SYSTEM furnace_naphtha_cracker
  (* Version 1.0, 2021-03-12, Lenovo *)
  APPLICATION furnace_naphtha_crackerApp
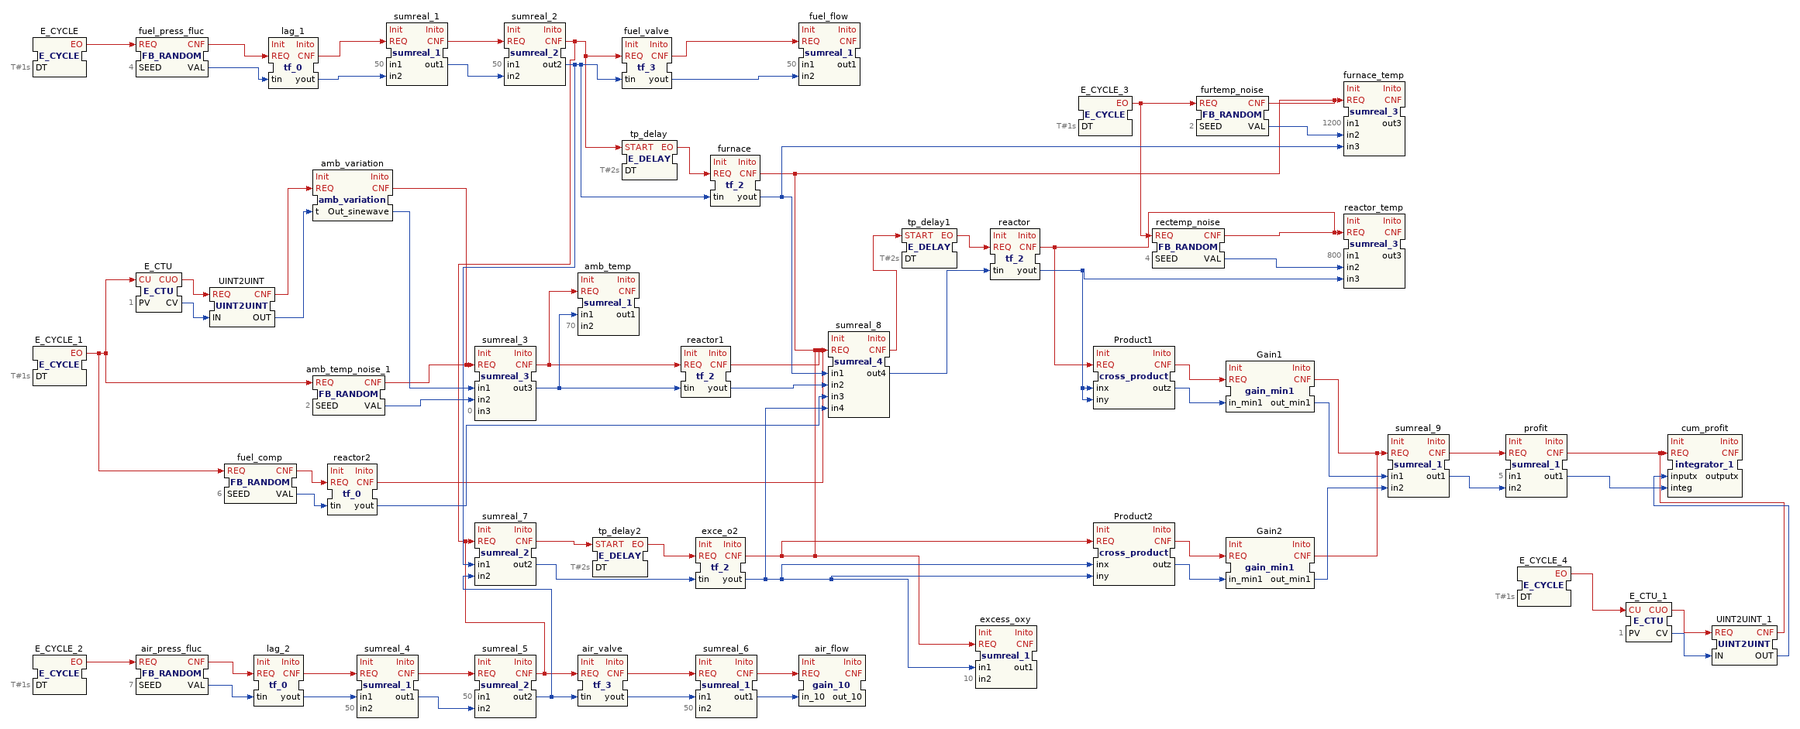
    FBS
      E_CYCLE : E_CYCLE(DT := T#1s);
      sumreal_1 : sumreal_1(in1 := 50);
      sumreal_2 : sumreal_2(in1 := 50);
      fuel_valve : tf_3;
      fuel_flow : sumreal_1(in1 := 50);
      E_CYCLE_1 : E_CYCLE(DT := T#1s);
      E_CTU : E_CTU(PV := 1);
      UINT2UINT : UINT2UINT;
      amb_variation : amb_variation;
      amb_temp_noise_1 : FB_RANDOM(SEED := 2);
      E_CYCLE_2 : E_CYCLE(DT := T#1s);
      air_press_fluc : FB_RANDOM(SEED := 7);
      lag_2 : tf_0;
      sumreal_4 : sumreal_1(in2 := 50);
      sumreal_5 : sumreal_2(in1 := 50);
      air_valve : tf_3;
      sumreal_6 : sumreal_1(in2 := 50);
      air_flow : gain_10;
      reactor1 : tf_2;
      fuel_comp : FB_RANDOM(SEED := 6);
      reactor2 : tf_0;
      sumreal_7 : sumreal_2;
      exce_o2 : tf_2;
      tp_delay : E_DELAY(DT := T#2s);
      furnace : tf_2;
      tp_delay2 : E_DELAY(DT := T#2s);
      sumreal_8 : sumreal_4;
      tp_delay1 : E_DELAY(DT := T#2s);
      reactor : tf_2;
      Product2 : cross_product;
      Gain2 : gain_min1;
      Product1 : cross_product;
      Gain1 : gain_min1;
      sumreal_9 : sumreal_1;
      E_CYCLE_3 : E_CYCLE(DT := T#1s);
      furtemp_noise : FB_RANDOM(SEED := 2);
      rectemp_noise : FB_RANDOM(SEED := 4);
      furnace_temp : sumreal_3(in1 := 1200);
      reactor_temp : sumreal_3(in1 := 800);
      profit : sumreal_1(in1 := 5);
      excess_oxy : sumreal_1(in2 := 10);
      E_CYCLE_4 : E_CYCLE(DT := T#1s);
      E_CTU_1 : E_CTU(PV := 1);
      UINT2UINT_1 : UINT2UINT;
      fuel_press_fluc : FB_RANDOM(SEED := 4);
      lag_1 : tf_0;
      sumreal_3 : sumreal_3(in3 := 0);
      amb_temp : sumreal_1(in2 := 70);
      cum_profit : integrator_1;
    END_FBS
    EVENT_CONNECTIONS
      sumreal_2.CNF TO fuel_valve.REQ;
      sumreal_1.CNF TO sumreal_2.REQ;
      fuel_valve.CNF TO fuel_flow.REQ;
      E_CYCLE_1.EO TO E_CTU.CU;
      E_CTU.CUO TO UINT2UINT.REQ;
      UINT2UINT.CNF TO amb_variation.REQ;
      E_CYCLE_1.EO TO amb_temp_noise_1.REQ;
      E_CYCLE_2.EO TO air_press_fluc.REQ;
      air_press_fluc.CNF TO lag_2.REQ;
      lag_2.CNF TO sumreal_4.REQ;
      sumreal_4.CNF TO sumreal_5.REQ;
      sumreal_5.CNF TO air_valve.REQ;
      air_valve.CNF TO sumreal_6.REQ;
      sumreal_6.CNF TO air_flow.REQ;
      E_CYCLE_1.EO TO fuel_comp.REQ;
      fuel_comp.CNF TO reactor2.REQ;
      sumreal_5.CNF TO sumreal_7.REQ;
      sumreal_2.CNF TO sumreal_7.REQ;
      sumreal_2.CNF TO tp_delay.START;
      tp_delay.EO TO furnace.REQ;
      sumreal_7.CNF TO tp_delay2.START;
      tp_delay2.EO TO exce_o2.REQ;
      furnace.CNF TO sumreal_8.REQ;
      reactor1.CNF TO sumreal_8.REQ;
      exce_o2.CNF TO sumreal_8.REQ;
      reactor2.CNF TO sumreal_8.REQ;
      sumreal_8.CNF TO tp_delay1.START;
      tp_delay1.EO TO reactor.REQ;
      exce_o2.CNF TO Product2.REQ;
      Product2.CNF TO Gain2.REQ;
      Product1.CNF TO Gain1.REQ;
      Gain1.CNF TO sumreal_9.REQ;
      Gain2.CNF TO sumreal_9.REQ;
      E_CYCLE_3.EO TO furtemp_noise.REQ;
      furnace.CNF TO furnace_temp.REQ;
      furtemp_noise.CNF TO furnace_temp.REQ;
      E_CYCLE_3.EO TO rectemp_noise.REQ;
      rectemp_noise.CNF TO reactor_temp.REQ;
      reactor.CNF TO Product1.REQ;
      reactor.CNF TO reactor_temp.REQ;
      sumreal_9.CNF TO profit.REQ;
      exce_o2.CNF TO excess_oxy.REQ;
      E_CTU_1.CUO TO UINT2UINT_1.REQ;
      E_CYCLE_4.EO TO E_CTU_1.CU;
      lag_1.CNF TO sumreal_1.REQ;
      E_CYCLE.EO TO fuel_press_fluc.REQ;
      fuel_press_fluc.CNF TO lag_1.REQ;
      sumreal_3.CNF TO reactor1.REQ;
      amb_temp_noise_1.CNF TO sumreal_3.REQ;
      amb_variation.CNF TO sumreal_3.REQ;
      sumreal_3.CNF TO amb_temp.REQ;
      profit.CNF TO cum_profit.REQ;
      UINT2UINT_1.CNF TO cum_profit.REQ;
    END_CONNECTIONS
    DATA_CONNECTIONS
      sumreal_1.out1 TO sumreal_2.in2;
      sumreal_2.out2 TO fuel_valve.tin;
      fuel_valve.yout TO fuel_flow.in2;
      E_CTU.CV TO UINT2UINT.IN;
      UINT2UINT.OUT TO amb_variation.t;
      air_press_fluc.VAL TO lag_2.tin;
      lag_2.yout TO sumreal_4.in1;
      sumreal_4.out1 TO sumreal_5.in2;
      sumreal_5.out2 TO air_valve.tin;
      air_valve.yout TO sumreal_6.in1;
      sumreal_6.out1 TO air_flow.in_10;
      fuel_comp.VAL TO reactor2.tin;
      sumreal_5.out2 TO sumreal_7.in2;
      sumreal_2.out2 TO sumreal_7.in1;
      sumreal_7.out2 TO exce_o2.tin;
      sumreal_2.out2 TO furnace.tin;
      furnace.yout TO sumreal_8.in1;
      reactor1.yout TO sumreal_8.in2;
      exce_o2.yout TO sumreal_8.in4;
      reactor2.yout TO sumreal_8.in3;
      sumreal_8.out4 TO reactor.tin;
      exce_o2.yout TO Product2.inx;
      exce_o2.yout TO Product2.iny;
      Product2.outz TO Gain2.in_min1;
      Product1.outz TO Gain1.in_min1;
      reactor.yout TO Product1.inx;
      reactor.yout TO Product1.iny;
      Gain2.out_min1 TO sumreal_9.in2;
      Gain1.out_min1 TO sumreal_9.in1;
      furtemp_noise.VAL TO furnace_temp.in2;
      furnace.yout TO furnace_temp.in3;
      rectemp_noise.VAL TO reactor_temp.in2;
      reactor.yout TO reactor_temp.in3;
      sumreal_9.out1 TO profit.in2;
      exce_o2.yout TO excess_oxy.in1;
      E_CTU_1.CV TO UINT2UINT_1.IN;
      lag_1.yout TO sumreal_1.in2;
      fuel_press_fluc.VAL TO lag_1.tin;
      sumreal_3.out3 TO reactor1.tin;
      amb_temp_noise_1.VAL TO sumreal_3.in2;
      amb_variation.Out_sinewave TO sumreal_3.in1;
      sumreal_3.out3 TO amb_temp.in1;
      UINT2UINT_1.OUT TO cum_profit.inputx;
      profit.out1 TO cum_profit.integ;
    END_CONNECTIONS
  END_APPLICATION
  DEVICE FORTE_PC : FORTE_PC(MGR_ID := "localhost:61499")
    {SET_ATTRIBUTE(Profile, HOLOBLOC)} (* device profile *)
    RESOURCE EMB_RES : EMB_RES
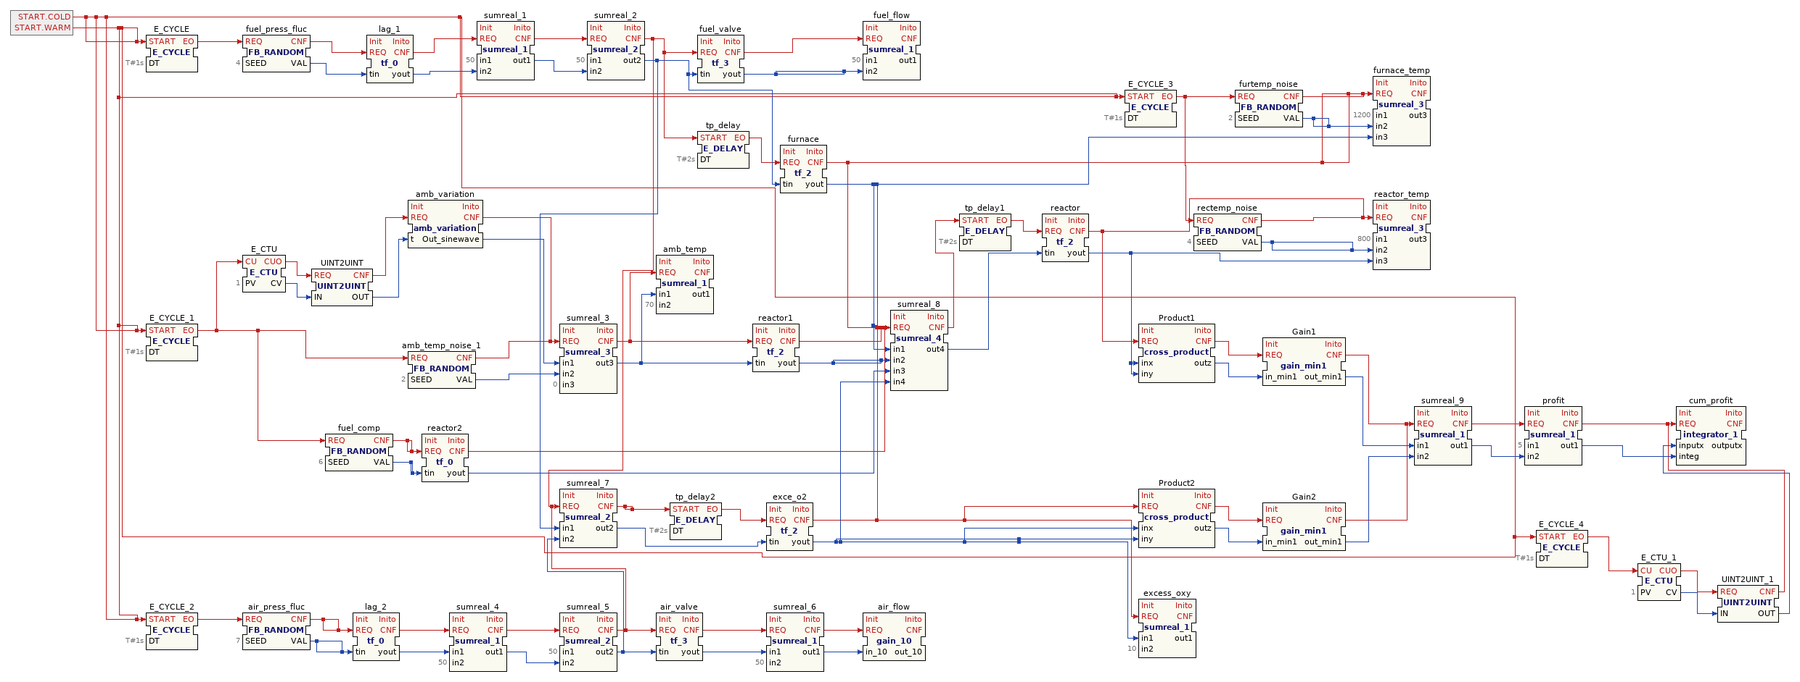
      FBS
        fuel_valve : tf_3;
        fuel_flow : sumreal_1(in1 := 50);
        E_CYCLE_1 : E_CYCLE(DT := T#1s);
        E_CTU : E_CTU(PV := 1);
        UINT2UINT : UINT2UINT;
        amb_variation : amb_variation;
        amb_temp_noise_1 : FB_RANDOM(SEED := 2);
        E_CYCLE_2 : E_CYCLE(DT := T#1s);
        air_press_fluc : FB_RANDOM(SEED := 7);
        lag_2 : tf_0;
        sumreal_4 : sumreal_1(in2 := 50);
        sumreal_5 : sumreal_2(in1 := 50);
        air_valve : tf_3;
        sumreal_6 : sumreal_1(in2 := 50);
        air_flow : gain_10;
        reactor1 : tf_2;
        fuel_comp : FB_RANDOM(SEED := 6);
        reactor2 : tf_0;
        sumreal_7 : sumreal_2;
        exce_o2 : tf_2;
        tp_delay : E_DELAY(DT := T#2s);
        furnace : tf_2;
        tp_delay2 : E_DELAY(DT := T#2s);
        sumreal_8 : sumreal_4;
        tp_delay1 : E_DELAY(DT := T#2s);
        reactor : tf_2;
        Product2 : cross_product;
        Gain2 : gain_min1;
        Product1 : cross_product;
        Gain1 : gain_min1;
        sumreal_9 : sumreal_1;
        E_CYCLE_3 : E_CYCLE(DT := T#1s);
        furtemp_noise : FB_RANDOM(SEED := 2);
        rectemp_noise : FB_RANDOM(SEED := 4);
        furnace_temp : sumreal_3(in1 := 1200);
        reactor_temp : sumreal_3(in1 := 800);
        profit : sumreal_1(in1 := 5);
        excess_oxy : sumreal_1(in2 := 10);
        E_CYCLE_4 : E_CYCLE(DT := T#1s);
        E_CTU_1 : E_CTU(PV := 1);
        UINT2UINT_1 : UINT2UINT;
        E_CYCLE : E_CYCLE(DT := T#1s);
        sumreal_1 : sumreal_1(in1 := 50);
        sumreal_2 : sumreal_2(in1 := 50);
        fuel_valve : tf_3;
        fuel_flow : sumreal_1(in1 := 50);
        E_CYCLE_1 : E_CYCLE(DT := T#1s);
        E_CTU : E_CTU(PV := 1);
        UINT2UINT : UINT2UINT;
        amb_variation : amb_variation;
        amb_temp_noise_1 : FB_RANDOM(SEED := 2);
        E_CYCLE_2 : E_CYCLE(DT := T#1s);
        air_press_fluc : FB_RANDOM(SEED := 7);
        lag_2 : tf_0;
        sumreal_4 : sumreal_1(in2 := 50);
        sumreal_5 : sumreal_2(in1 := 50);
        air_valve : tf_3;
        sumreal_6 : sumreal_1(in2 := 50);
        air_flow : gain_10;
        reactor1 : tf_2;
        fuel_comp : FB_RANDOM(SEED := 6);
        reactor2 : tf_0;
        sumreal_7 : sumreal_2;
        exce_o2 : tf_2;
        tp_delay : E_DELAY(DT := T#2s);
        furnace : tf_2;
        tp_delay2 : E_DELAY(DT := T#2s);
        sumreal_8 : sumreal_4;
        tp_delay1 : E_DELAY(DT := T#2s);
        reactor : tf_2;
        Product2 : cross_product;
        Gain2 : gain_min1;
        Product1 : cross_product;
        Gain1 : gain_min1;
        sumreal_9 : sumreal_1;
        E_CYCLE_3 : E_CYCLE(DT := T#1s);
        furtemp_noise : FB_RANDOM(SEED := 2);
        rectemp_noise : FB_RANDOM(SEED := 4);
        furnace_temp : sumreal_3(in1 := 1200);
        reactor_temp : sumreal_3(in1 := 800);
        profit : sumreal_1(in1 := 5);
        excess_oxy : sumreal_1(in2 := 10);
        E_CYCLE_4 : E_CYCLE(DT := T#1s);
        E_CTU_1 : E_CTU(PV := 1);
        UINT2UINT_1 : UINT2UINT;
        fuel_press_fluc : FB_RANDOM(SEED := 4);
        lag_1 : tf_0;
        sumreal_3 : sumreal_3(in3 := 0);
        amb_temp : sumreal_1(in2 := 70);
        cum_profit : integrator_1;
        sumreal_2 : sumreal_2(in1 := 50);
        sumreal_1 : sumreal_1(in1 := 50);
        E_CYCLE : E_CYCLE(DT := T#1s);
      END_FBS
      EVENT_CONNECTIONS
        fuel_valve.CNF TO fuel_flow.REQ;
        E_CYCLE_1.EO TO E_CTU.CU;
        E_CTU.CUO TO UINT2UINT.REQ;
        UINT2UINT.CNF TO amb_variation.REQ;
        E_CYCLE_1.EO TO amb_temp_noise_1.REQ;
        E_CYCLE_2.EO TO air_press_fluc.REQ;
        air_press_fluc.CNF TO lag_2.REQ;
        lag_2.CNF TO sumreal_4.REQ;
        sumreal_4.CNF TO sumreal_5.REQ;
        sumreal_5.CNF TO air_valve.REQ;
        air_valve.CNF TO sumreal_6.REQ;
        sumreal_6.CNF TO air_flow.REQ;
        E_CYCLE_1.EO TO fuel_comp.REQ;
        fuel_comp.CNF TO reactor2.REQ;
        sumreal_5.CNF TO sumreal_7.REQ;
        tp_delay.EO TO furnace.REQ;
        sumreal_7.CNF TO tp_delay2.START;
        tp_delay2.EO TO exce_o2.REQ;
        furnace.CNF TO sumreal_8.REQ;
        reactor1.CNF TO sumreal_8.REQ;
        exce_o2.CNF TO sumreal_8.REQ;
        reactor2.CNF TO sumreal_8.REQ;
        sumreal_8.CNF TO tp_delay1.START;
        tp_delay1.EO TO reactor.REQ;
        exce_o2.CNF TO Product2.REQ;
        Product2.CNF TO Gain2.REQ;
        reactor.CNF TO Product1.REQ;
        Product1.CNF TO Gain1.REQ;
        Gain1.CNF TO sumreal_9.REQ;
        Gain2.CNF TO sumreal_9.REQ;
        E_CYCLE_3.EO TO furtemp_noise.REQ;
        E_CYCLE_3.EO TO rectemp_noise.REQ;
        furnace.CNF TO furnace_temp.REQ;
        furtemp_noise.CNF TO furnace_temp.REQ;
        rectemp_noise.CNF TO reactor_temp.REQ;
        reactor.CNF TO reactor_temp.REQ;
        sumreal_9.CNF TO profit.REQ;
        exce_o2.CNF TO excess_oxy.REQ;
        E_CYCLE_4.EO TO E_CTU_1.CU;
        E_CTU_1.CUO TO UINT2UINT_1.REQ;
        sumreal_1.CNF TO sumreal_2.REQ;
        sumreal_2.CNF TO fuel_valve.REQ;
        fuel_valve.CNF TO fuel_flow.REQ;
        E_CYCLE_1.EO TO E_CTU.CU;
        E_CTU.CUO TO UINT2UINT.REQ;
        UINT2UINT.CNF TO amb_variation.REQ;
        E_CYCLE_1.EO TO amb_temp_noise_1.REQ;
        E_CYCLE_2.EO TO air_press_fluc.REQ;
        air_press_fluc.CNF TO lag_2.REQ;
        lag_2.CNF TO sumreal_4.REQ;
        sumreal_4.CNF TO sumreal_5.REQ;
        sumreal_5.CNF TO air_valve.REQ;
        air_valve.CNF TO sumreal_6.REQ;
        sumreal_6.CNF TO air_flow.REQ;
        E_CYCLE_1.EO TO fuel_comp.REQ;
        fuel_comp.CNF TO reactor2.REQ;
        sumreal_5.CNF TO sumreal_7.REQ;
        sumreal_2.CNF TO sumreal_7.REQ;
        sumreal_2.CNF TO tp_delay.START;
        tp_delay.EO TO furnace.REQ;
        sumreal_7.CNF TO tp_delay2.START;
        tp_delay2.EO TO exce_o2.REQ;
        furnace.CNF TO sumreal_8.REQ;
        reactor1.CNF TO sumreal_8.REQ;
        exce_o2.CNF TO sumreal_8.REQ;
        reactor2.CNF TO sumreal_8.REQ;
        sumreal_8.CNF TO tp_delay1.START;
        tp_delay1.EO TO reactor.REQ;
        exce_o2.CNF TO Product2.REQ;
        Product2.CNF TO Gain2.REQ;
        reactor.CNF TO Product1.REQ;
        Product1.CNF TO Gain1.REQ;
        Gain1.CNF TO sumreal_9.REQ;
        Gain2.CNF TO sumreal_9.REQ;
        E_CYCLE_3.EO TO furtemp_noise.REQ;
        E_CYCLE_3.EO TO rectemp_noise.REQ;
        furnace.CNF TO furnace_temp.REQ;
        furtemp_noise.CNF TO furnace_temp.REQ;
        rectemp_noise.CNF TO reactor_temp.REQ;
        reactor.CNF TO reactor_temp.REQ;
        sumreal_9.CNF TO profit.REQ;
        exce_o2.CNF TO excess_oxy.REQ;
        E_CYCLE_4.EO TO E_CTU_1.CU;
        E_CTU_1.CUO TO UINT2UINT_1.REQ;
        E_CYCLE.EO TO fuel_press_fluc.REQ;
        fuel_press_fluc.CNF TO lag_1.REQ;
        lag_1.CNF TO sumreal_1.REQ;
        amb_temp_noise_1.CNF TO sumreal_3.REQ;
        amb_variation.CNF TO sumreal_3.REQ;
        sumreal_3.CNF TO reactor1.REQ;
        sumreal_3.CNF TO amb_temp.REQ;
        profit.CNF TO cum_profit.REQ;
        UINT2UINT_1.CNF TO cum_profit.REQ;
        START.COLD TO E_CYCLE.START;
        START.WARM TO E_CYCLE.START;
        START.COLD TO E_CYCLE_1.START;
        START.WARM TO E_CYCLE_1.START;
        START.COLD TO E_CYCLE_2.START;
        START.WARM TO E_CYCLE_2.START;
        START.COLD TO E_CYCLE_4.START;
        START.WARM TO E_CYCLE_4.START;
        START.COLD TO E_CYCLE_3.START;
        START.WARM TO E_CYCLE_3.START;
        sumreal_2.CNF TO tp_delay.START;
        sumreal_2.CNF TO sumreal_7.REQ;
        sumreal_2.CNF TO fuel_valve.REQ;
        sumreal_1.CNF TO sumreal_2.REQ;
      END_CONNECTIONS
      DATA_CONNECTIONS
        fuel_valve.yout TO fuel_flow.in2;
        E_CTU.CV TO UINT2UINT.IN;
        UINT2UINT.OUT TO amb_variation.t;
        air_press_fluc.VAL TO lag_2.tin;
        lag_2.yout TO sumreal_4.in1;
        sumreal_4.out1 TO sumreal_5.in2;
        sumreal_5.out2 TO air_valve.tin;
        air_valve.yout TO sumreal_6.in1;
        sumreal_6.out1 TO air_flow.in_10;
        fuel_comp.VAL TO reactor2.tin;
        sumreal_5.out2 TO sumreal_7.in2;
        sumreal_7.out2 TO exce_o2.tin;
        furnace.yout TO sumreal_8.in1;
        reactor1.yout TO sumreal_8.in2;
        reactor2.yout TO sumreal_8.in3;
        exce_o2.yout TO sumreal_8.in4;
        sumreal_8.out4 TO reactor.tin;
        exce_o2.yout TO Product2.inx;
        exce_o2.yout TO Product2.iny;
        Product2.outz TO Gain2.in_min1;
        reactor.yout TO Product1.inx;
        reactor.yout TO Product1.iny;
        Product1.outz TO Gain1.in_min1;
        Gain1.out_min1 TO sumreal_9.in1;
        Gain2.out_min1 TO sumreal_9.in2;
        furtemp_noise.VAL TO furnace_temp.in2;
        furnace.yout TO furnace_temp.in3;
        rectemp_noise.VAL TO reactor_temp.in2;
        reactor.yout TO reactor_temp.in3;
        sumreal_9.out1 TO profit.in2;
        exce_o2.yout TO excess_oxy.in1;
        E_CTU_1.CV TO UINT2UINT_1.IN;
        sumreal_1.out1 TO sumreal_2.in2;
        sumreal_2.out2 TO fuel_valve.tin;
        fuel_valve.yout TO fuel_flow.in2;
        E_CTU.CV TO UINT2UINT.IN;
        UINT2UINT.OUT TO amb_variation.t;
        air_press_fluc.VAL TO lag_2.tin;
        lag_2.yout TO sumreal_4.in1;
        sumreal_4.out1 TO sumreal_5.in2;
        sumreal_5.out2 TO air_valve.tin;
        air_valve.yout TO sumreal_6.in1;
        sumreal_6.out1 TO air_flow.in_10;
        fuel_comp.VAL TO reactor2.tin;
        sumreal_2.out2 TO sumreal_7.in1;
        sumreal_5.out2 TO sumreal_7.in2;
        sumreal_7.out2 TO exce_o2.tin;
        sumreal_2.out2 TO furnace.tin;
        furnace.yout TO sumreal_8.in1;
        reactor1.yout TO sumreal_8.in2;
        reactor2.yout TO sumreal_8.in3;
        exce_o2.yout TO sumreal_8.in4;
        sumreal_8.out4 TO reactor.tin;
        exce_o2.yout TO Product2.inx;
        exce_o2.yout TO Product2.iny;
        Product2.outz TO Gain2.in_min1;
        reactor.yout TO Product1.inx;
        reactor.yout TO Product1.iny;
        Product1.outz TO Gain1.in_min1;
        Gain1.out_min1 TO sumreal_9.in1;
        Gain2.out_min1 TO sumreal_9.in2;
        furtemp_noise.VAL TO furnace_temp.in2;
        furnace.yout TO furnace_temp.in3;
        rectemp_noise.VAL TO reactor_temp.in2;
        reactor.yout TO reactor_temp.in3;
        sumreal_9.out1 TO profit.in2;
        exce_o2.yout TO excess_oxy.in1;
        E_CTU_1.CV TO UINT2UINT_1.IN;
        fuel_press_fluc.VAL TO lag_1.tin;
        lag_1.yout TO sumreal_1.in2;
        amb_variation.Out_sinewave TO sumreal_3.in1;
        amb_temp_noise_1.VAL TO sumreal_3.in2;
        sumreal_3.out3 TO reactor1.tin;
        sumreal_3.out3 TO amb_temp.in1;
        UINT2UINT_1.OUT TO cum_profit.inputx;
        profit.out1 TO cum_profit.integ;
        sumreal_2.out2 TO furnace.tin;
        sumreal_2.out2 TO sumreal_7.in1;
        sumreal_2.out2 TO fuel_valve.tin;
        sumreal_1.out1 TO sumreal_2.in2;
      END_CONNECTIONS
    END_RESOURCE
  END_DEVICE
  MAPPINGS
    furnace_naphtha_crackerApp.fuel_valve ON FORTE_PC.EMB_RES.fuel_valve;
    furnace_naphtha_crackerApp.fuel_flow ON FORTE_PC.EMB_RES.fuel_flow;
    furnace_naphtha_crackerApp.E_CYCLE_1 ON FORTE_PC.EMB_RES.E_CYCLE_1;
    furnace_naphtha_crackerApp.E_CTU ON FORTE_PC.EMB_RES.E_CTU;
    furnace_naphtha_crackerApp.UINT2UINT ON FORTE_PC.EMB_RES.UINT2UINT;
    furnace_naphtha_crackerApp.amb_variation ON FORTE_PC.EMB_RES.amb_variation;
    furnace_naphtha_crackerApp.amb_temp_noise_1 ON FORTE_PC.EMB_RES.amb_temp_noise_1;
    furnace_naphtha_crackerApp.E_CYCLE_2 ON FORTE_PC.EMB_RES.E_CYCLE_2;
    furnace_naphtha_crackerApp.air_press_fluc ON FORTE_PC.EMB_RES.air_press_fluc;
    furnace_naphtha_crackerApp.lag_2 ON FORTE_PC.EMB_RES.lag_2;
    furnace_naphtha_crackerApp.sumreal_4 ON FORTE_PC.EMB_RES.sumreal_4;
    furnace_naphtha_crackerApp.sumreal_5 ON FORTE_PC.EMB_RES.sumreal_5;
    furnace_naphtha_crackerApp.air_valve ON FORTE_PC.EMB_RES.air_valve;
    furnace_naphtha_crackerApp.sumreal_6 ON FORTE_PC.EMB_RES.sumreal_6;
    furnace_naphtha_crackerApp.air_flow ON FORTE_PC.EMB_RES.air_flow;
    furnace_naphtha_crackerApp.reactor1 ON FORTE_PC.EMB_RES.reactor1;
    furnace_naphtha_crackerApp.fuel_comp ON FORTE_PC.EMB_RES.fuel_comp;
    furnace_naphtha_crackerApp.reactor2 ON FORTE_PC.EMB_RES.reactor2;
    furnace_naphtha_crackerApp.sumreal_7 ON FORTE_PC.EMB_RES.sumreal_7;
    furnace_naphtha_crackerApp.exce_o2 ON FORTE_PC.EMB_RES.exce_o2;
    furnace_naphtha_crackerApp.tp_delay ON FORTE_PC.EMB_RES.tp_delay;
    furnace_naphtha_crackerApp.furnace ON FORTE_PC.EMB_RES.furnace;
    furnace_naphtha_crackerApp.tp_delay2 ON FORTE_PC.EMB_RES.tp_delay2;
    furnace_naphtha_crackerApp.sumreal_8 ON FORTE_PC.EMB_RES.sumreal_8;
    furnace_naphtha_crackerApp.tp_delay1 ON FORTE_PC.EMB_RES.tp_delay1;
    furnace_naphtha_crackerApp.reactor ON FORTE_PC.EMB_RES.reactor;
    furnace_naphtha_crackerApp.Product2 ON FORTE_PC.EMB_RES.Product2;
    furnace_naphtha_crackerApp.Gain2 ON FORTE_PC.EMB_RES.Gain2;
    furnace_naphtha_crackerApp.Product1 ON FORTE_PC.EMB_RES.Product1;
    furnace_naphtha_crackerApp.Gain1 ON FORTE_PC.EMB_RES.Gain1;
    furnace_naphtha_crackerApp.sumreal_9 ON FORTE_PC.EMB_RES.sumreal_9;
    furnace_naphtha_crackerApp.E_CYCLE_3 ON FORTE_PC.EMB_RES.E_CYCLE_3;
    furnace_naphtha_crackerApp.furtemp_noise ON FORTE_PC.EMB_RES.furtemp_noise;
    furnace_naphtha_crackerApp.rectemp_noise ON FORTE_PC.EMB_RES.rectemp_noise;
    furnace_naphtha_crackerApp.furnace_temp ON FORTE_PC.EMB_RES.furnace_temp;
    furnace_naphtha_crackerApp.reactor_temp ON FORTE_PC.EMB_RES.reactor_temp;
    furnace_naphtha_crackerApp.profit ON FORTE_PC.EMB_RES.profit;
    furnace_naphtha_crackerApp.excess_oxy ON FORTE_PC.EMB_RES.excess_oxy;
    furnace_naphtha_crackerApp.E_CYCLE_4 ON FORTE_PC.EMB_RES.E_CYCLE_4;
    furnace_naphtha_crackerApp.E_CTU_1 ON FORTE_PC.EMB_RES.E_CTU_1;
    furnace_naphtha_crackerApp.UINT2UINT_1 ON FORTE_PC.EMB_RES.UINT2UINT_1;
    furnace_naphtha_crackerApp.E_CYCLE ON FORTE_PC.EMB_RES.E_CYCLE;
    furnace_naphtha_crackerApp.sumreal_1 ON FORTE_PC.EMB_RES.sumreal_1;
    furnace_naphtha_crackerApp.sumreal_2 ON FORTE_PC.EMB_RES.sumreal_2;
    furnace_naphtha_crackerApp.fuel_valve ON FORTE_PC.EMB_RES.fuel_valve;
    furnace_naphtha_crackerApp.fuel_flow ON FORTE_PC.EMB_RES.fuel_flow;
    furnace_naphtha_crackerApp.E_CYCLE_1 ON FORTE_PC.EMB_RES.E_CYCLE_1;
    furnace_naphtha_crackerApp.E_CTU ON FORTE_PC.EMB_RES.E_CTU;
    furnace_naphtha_crackerApp.UINT2UINT ON FORTE_PC.EMB_RES.UINT2UINT;
    furnace_naphtha_crackerApp.amb_variation ON FORTE_PC.EMB_RES.amb_variation;
    furnace_naphtha_crackerApp.amb_temp_noise_1 ON FORTE_PC.EMB_RES.amb_temp_noise_1;
    furnace_naphtha_crackerApp.E_CYCLE_2 ON FORTE_PC.EMB_RES.E_CYCLE_2;
    furnace_naphtha_crackerApp.air_press_fluc ON FORTE_PC.EMB_RES.air_press_fluc;
    furnace_naphtha_crackerApp.lag_2 ON FORTE_PC.EMB_RES.lag_2;
    furnace_naphtha_crackerApp.sumreal_4 ON FORTE_PC.EMB_RES.sumreal_4;
    furnace_naphtha_crackerApp.sumreal_5 ON FORTE_PC.EMB_RES.sumreal_5;
    furnace_naphtha_crackerApp.air_valve ON FORTE_PC.EMB_RES.air_valve;
    furnace_naphtha_crackerApp.sumreal_6 ON FORTE_PC.EMB_RES.sumreal_6;
    furnace_naphtha_crackerApp.air_flow ON FORTE_PC.EMB_RES.air_flow;
    furnace_naphtha_crackerApp.reactor1 ON FORTE_PC.EMB_RES.reactor1;
    furnace_naphtha_crackerApp.fuel_comp ON FORTE_PC.EMB_RES.fuel_comp;
    furnace_naphtha_crackerApp.reactor2 ON FORTE_PC.EMB_RES.reactor2;
    furnace_naphtha_crackerApp.sumreal_7 ON FORTE_PC.EMB_RES.sumreal_7;
    furnace_naphtha_crackerApp.exce_o2 ON FORTE_PC.EMB_RES.exce_o2;
    furnace_naphtha_crackerApp.tp_delay ON FORTE_PC.EMB_RES.tp_delay;
    furnace_naphtha_crackerApp.furnace ON FORTE_PC.EMB_RES.furnace;
    furnace_naphtha_crackerApp.tp_delay2 ON FORTE_PC.EMB_RES.tp_delay2;
    furnace_naphtha_crackerApp.sumreal_8 ON FORTE_PC.EMB_RES.sumreal_8;
    furnace_naphtha_crackerApp.tp_delay1 ON FORTE_PC.EMB_RES.tp_delay1;
    furnace_naphtha_crackerApp.reactor ON FORTE_PC.EMB_RES.reactor;
    furnace_naphtha_crackerApp.Product2 ON FORTE_PC.EMB_RES.Product2;
    furnace_naphtha_crackerApp.Gain2 ON FORTE_PC.EMB_RES.Gain2;
    furnace_naphtha_crackerApp.Product1 ON FORTE_PC.EMB_RES.Product1;
    furnace_naphtha_crackerApp.Gain1 ON FORTE_PC.EMB_RES.Gain1;
    furnace_naphtha_crackerApp.sumreal_9 ON FORTE_PC.EMB_RES.sumreal_9;
    furnace_naphtha_crackerApp.E_CYCLE_3 ON FORTE_PC.EMB_RES.E_CYCLE_3;
    furnace_naphtha_crackerApp.furtemp_noise ON FORTE_PC.EMB_RES.furtemp_noise;
    furnace_naphtha_crackerApp.rectemp_noise ON FORTE_PC.EMB_RES.rectemp_noise;
    furnace_naphtha_crackerApp.furnace_temp ON FORTE_PC.EMB_RES.furnace_temp;
    furnace_naphtha_crackerApp.reactor_temp ON FORTE_PC.EMB_RES.reactor_temp;
    furnace_naphtha_crackerApp.profit ON FORTE_PC.EMB_RES.profit;
    furnace_naphtha_crackerApp.excess_oxy ON FORTE_PC.EMB_RES.excess_oxy;
    furnace_naphtha_crackerApp.E_CYCLE_4 ON FORTE_PC.EMB_RES.E_CYCLE_4;
    furnace_naphtha_crackerApp.E_CTU_1 ON FORTE_PC.EMB_RES.E_CTU_1;
    furnace_naphtha_crackerApp.UINT2UINT_1 ON FORTE_PC.EMB_RES.UINT2UINT_1;
    furnace_naphtha_crackerApp.fuel_press_fluc ON FORTE_PC.EMB_RES.fuel_press_fluc;
    furnace_naphtha_crackerApp.lag_1 ON FORTE_PC.EMB_RES.lag_1;
    furnace_naphtha_crackerApp.sumreal_3 ON FORTE_PC.EMB_RES.sumreal_3;
    furnace_naphtha_crackerApp.amb_temp ON FORTE_PC.EMB_RES.amb_temp;
    furnace_naphtha_crackerApp.cum_profit ON FORTE_PC.EMB_RES.cum_profit;
    furnace_naphtha_crackerApp.sumreal_2 ON FORTE_PC.EMB_RES.sumreal_2;
    furnace_naphtha_crackerApp.sumreal_1 ON FORTE_PC.EMB_RES.sumreal_1;
    furnace_naphtha_crackerApp.E_CYCLE ON FORTE_PC.EMB_RES.E_CYCLE;
  END_MAPPINGS
  SEGMENTS
    Ethernet : Ethernet;
  END_SEGMENTS
  LINKS
    FORTE_PC => Ethernet;
  END_LINKS
END_SYSTEM
